// LS Electric XG5000 project: 과년69_1
// PLC NewPLC
// module base 0 slot 0: 입출력 모듈:XBC-DR20S (DC 24V 입력 12점, 릴레이 출력 8점)

PROGRAM NewProgram (task: 스캔 프로그램)

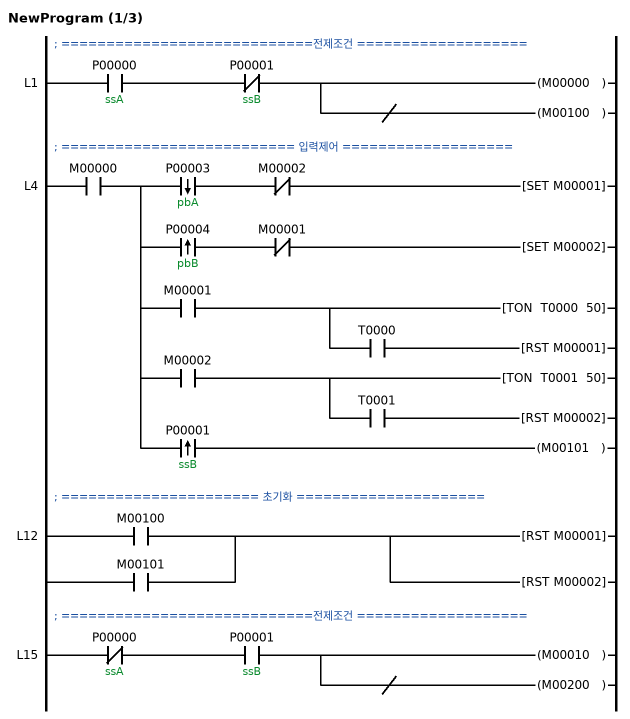
// ============================전제조건 ===================
; L1
LOAD      P00000	// ssA
AND NOT   P00001	// ssB
OUT       M00000
NOT
OUT       M00100
// ========================== 입력제어 ===================
; L4
LOAD      M00000
MPUSH
ANDN      P00003	// pbA
AND NOT   M00002
SET       M00001
MLOAD
ANDP      P00004	// pbB
AND NOT   M00001
SET       M00002
MLOAD
AND       M00001
TON       T0000 50
AND       T0000
RST       M00001
MLOAD
AND       M00002
TON       T0001 50
AND       T0001
RST       M00002
MPOP
ANDP      P00001	// ssB
OUT       M00101
// ====================== 초기화 =====================
; L12
LOAD      M00100
OR        M00101
RST       M00001
RST       M00002
// ============================전제조건 ===================
; L15
LOAD NOT  P00000	// ssA
AND       P00001	// ssB
OUT       M00010
NOT
OUT       M00200

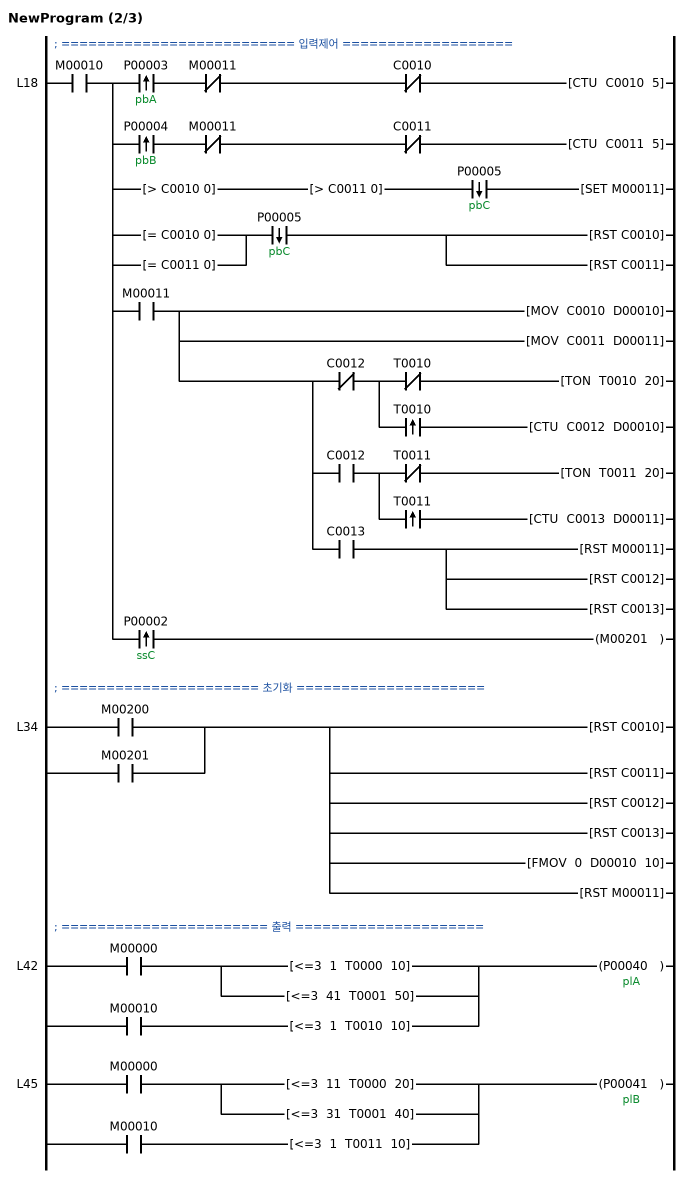
// ========================== 입력제어 ===================
; L18
LOAD      M00010
MPUSH
ANDP      P00003	// pbA
AND NOT   M00011
AND NOT   C0010
CTU       C0010 5
MLOAD
ANDP      P00004	// pbB
AND NOT   M00011
AND NOT   C0011
CTU       C0011 5
MLOAD
AND>      C0010 0
AND>      C0011 0
ANDN      P00005	// pbC
SET       M00011
MLOAD
LOAD=     C0010 0
OR=       C0011 0
AND LOAD
ANDN      P00005	// pbC
RST       C0010
RST       C0011
MLOAD
AND       M00011
MOV       C0010 D00010
MOV       C0011 D00011
MPUSH
AND NOT   C0012
MPUSH
AND NOT   T0010
TON       T0010 20
MPOP
ANDP      T0010
CTU       C0012 D00010
MLOAD
AND       C0012
MPUSH
AND NOT   T0011
TON       T0011 20
MPOP
ANDP      T0011
CTU       C0013 D00011
MPOP
AND       C0013
RST       M00011
RST       C0012
RST       C0013
MPOP
ANDP      P00002	// ssC
OUT       M00201
// ====================== 초기화 =====================
; L34
LOAD      M00200
OR        M00201
RST       C0010
RST       C0011
RST       C0012
RST       C0013
FMOV      0 D00010 10
RST       M00011
// ======================= 출력 =====================
; L42
LOAD      M00000
LOAD<=3   1 T0000 10
OR<=3     41 T0001 50
AND LOAD
LOAD      M00010
AND<=3    1 T0010 10
OR LOAD
OUT       P00040	// plA
; L45
LOAD      M00000
LOAD<=3   11 T0000 20
OR<=3     31 T0001 40
AND LOAD
LOAD      M00010
AND<=3    1 T0011 10
OR LOAD
OUT       P00041	// plB

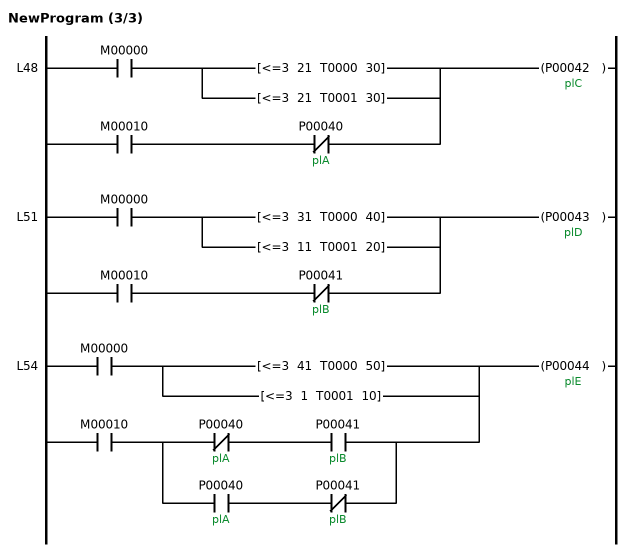
; L48
LOAD      M00000
LOAD<=3   21 T0000 30
OR<=3     21 T0001 30
AND LOAD
LOAD      M00010
AND NOT   P00040	// plA
OR LOAD
OUT       P00042	// plC
; L51
LOAD      M00000
LOAD<=3   31 T0000 40
OR<=3     11 T0001 20
AND LOAD
LOAD      M00010
AND NOT   P00041	// plB
OR LOAD
OUT       P00043	// plD
; L54
LOAD      M00000
LOAD<=3   41 T0000 50
OR<=3     1 T0001 10
AND LOAD
LOAD      M00010
LOAD NOT  P00040	// plA
AND       P00041	// plB
LOAD      P00040	// plA
AND NOT   P00041	// plB
OR LOAD
AND LOAD
OR LOAD
OUT       P00044	// plE